PROGRAM MAIN
VAR
END_VAR

END_PROGRAM

(* stored: Version 1.1.0.1
   POU MAIN: Id {13fc9eb7-def6-4e13-aac0-0e3df95d5012} *)
